TYPE ES_ALARM :
	STRUCT
		
		Enable			:BOOL;
		Active			:BOOL;
		Reset			:BOOL;
		tmr				:TON;
		pt				:INT:=7;		//secondi
		
	END_STRUCT
END_TYPE

(* stored: Version 1.1.0.1, ProductVersion 3.1.4022.12
   DUT ES_ALARM: Id {ea1e1d25-90ac-483e-8488-74c395af2e10} *)
